PROGRAM IO_OP10A_10B_JB
VAR
	//INPUT
	WORD_AS_BIT_0: WORD_AS_BIT;
	WORD_AS_BIT_1: WORD_AS_BIT;
	WORD_AS_BIT_2: WORD_AS_BIT;
	WORD_AS_BIT_3: WORD_AS_BIT;	
	//OUTPUT
	BIT_AS_WORD_0: BIT_AS_WORD;
	BIT_AS_WORD_1: BIT_AS_WORD;
	BIT_AS_WORD_2: BIT_AS_WORD;
	BIT_AS_WORD_3: BIT_AS_WORD;	
	//OP10A JB DI/DO 
	OP10A_BOWL_FEEDER_JB_16DI_MODULE_1 AT %I* : WORD;
	OP10A_BOWL_FEEDER_JB_16DI_MODULE_2 AT %I* : WORD;
	OP10A_BOWL_FEEDER_JB_16DO_MODULE_1 AT %Q* : WORD;
	OP10A_BOWL_FEEDER_JB_16DO_MODULE_2 AT %Q* : WORD;
	//OP10B JB DI/DO 
	OP10B_BOWL_FEEDER_JB_16DI_MODULE_1 AT %I* : WORD;
	OP10B_BOWL_FEEDER_JB_16DI_MODULE_2 AT %I* : WORD;
	OP10B_BOWL_FEEDER_JB_16DO_MODULE_1 AT %Q* : WORD;
	OP10B_BOWL_FEEDER_JB_16DO_MODULE_2 AT %Q* : WORD;
END_VAR

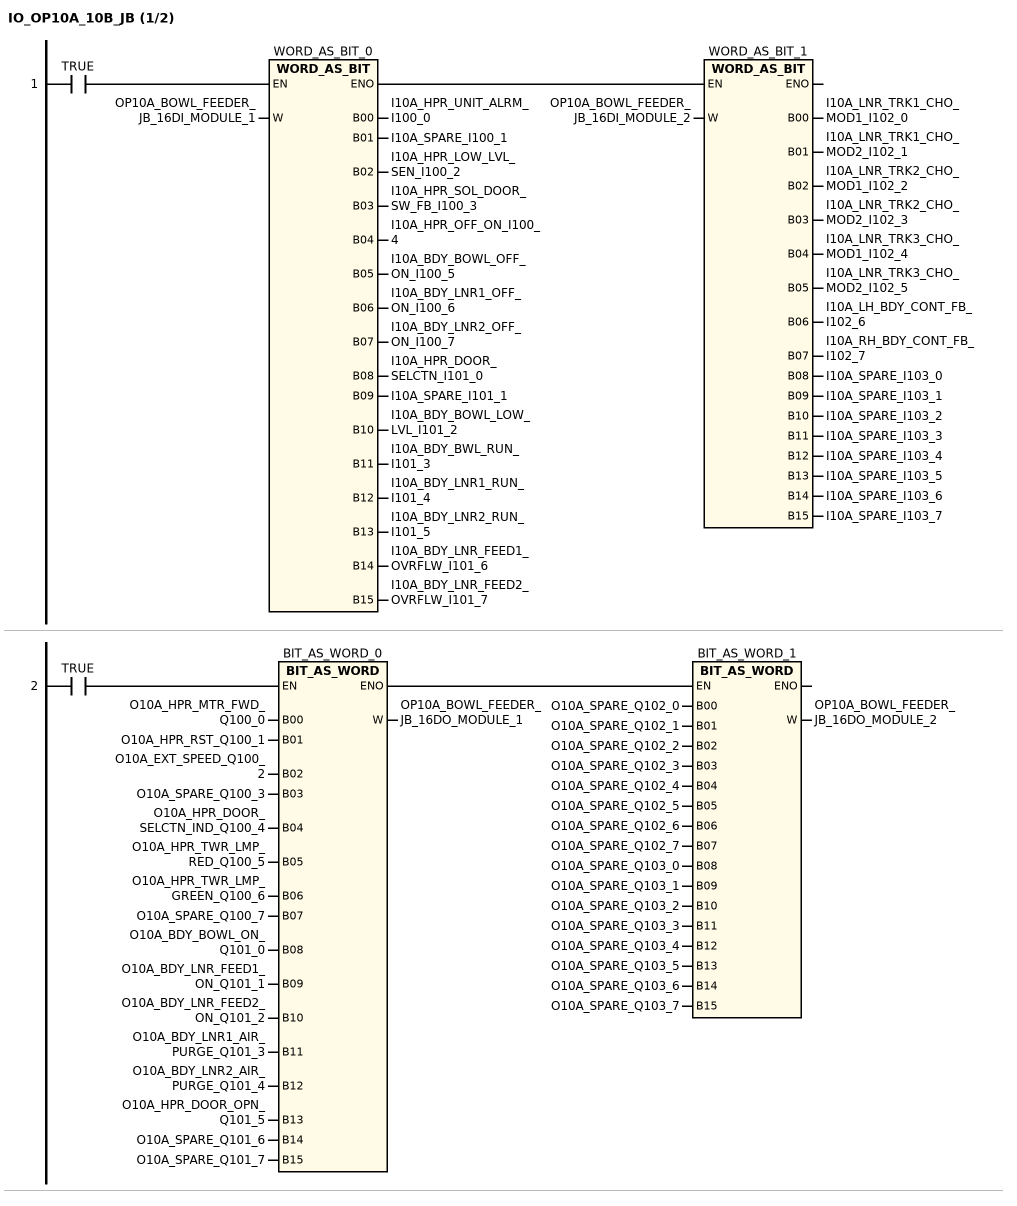
// NETWORK 1
WORD_AS_BIT_0(
    W := OP10A_BOWL_FEEDER_JB_16DI_MODULE_1,
    B00 => I10A_HPR_UNIT_ALRM_I100_0,
    B01 => I10A_SPARE_I100_1,
    B02 => I10A_HPR_LOW_LVL_SEN_I100_2,
    B03 => I10A_HPR_SOL_DOOR_SW_FB_I100_3,
    B04 => I10A_HPR_OFF_ON_I100_4,
    B05 => I10A_BDY_BOWL_OFF_ON_I100_5,
    B06 => I10A_BDY_LNR1_OFF_ON_I100_6,
    B07 => I10A_BDY_LNR2_OFF_ON_I100_7,
    B08 => I10A_HPR_DOOR_SELCTN_I101_0,
    B09 => I10A_SPARE_I101_1,
    B10 => I10A_BDY_BOWL_LOW_LVL_I101_2,
    B11 => I10A_BDY_BWL_RUN_I101_3,
    B12 => I10A_BDY_LNR1_RUN_I101_4,
    B13 => I10A_BDY_LNR2_RUN_I101_5,
    B14 => I10A_BDY_LNR_FEED1_OVRFLW_I101_6,
    B15 => I10A_BDY_LNR_FEED2_OVRFLW_I101_7); // WORD_AS_BIT
WORD_AS_BIT_1(
    W := OP10A_BOWL_FEEDER_JB_16DI_MODULE_2,
    B00 => I10A_LNR_TRK1_CHO_MOD1_I102_0,
    B01 => I10A_LNR_TRK1_CHO_MOD2_I102_1,
    B02 => I10A_LNR_TRK2_CHO_MOD1_I102_2,
    B03 => I10A_LNR_TRK2_CHO_MOD2_I102_3,
    B04 => I10A_LNR_TRK3_CHO_MOD1_I102_4,
    B05 => I10A_LNR_TRK3_CHO_MOD2_I102_5,
    B06 => I10A_LH_BDY_CONT_FB_I102_6,
    B07 => I10A_RH_BDY_CONT_FB_I102_7,
    B08 => I10A_SPARE_I103_0,
    B09 => I10A_SPARE_I103_1,
    B10 => I10A_SPARE_I103_2,
    B11 => I10A_SPARE_I103_3,
    B12 => I10A_SPARE_I103_4,
    B13 => I10A_SPARE_I103_5,
    B14 => I10A_SPARE_I103_6,
    B15 => I10A_SPARE_I103_7); // WORD_AS_BIT

// NETWORK 2
BIT_AS_WORD_0(
    B00 := O10A_HPR_MTR_FWD_Q100_0,
    B01 := O10A_HPR_RST_Q100_1,
    B02 := O10A_EXT_SPEED_Q100_2,
    B03 := O10A_SPARE_Q100_3,
    B04 := O10A_HPR_DOOR_SELCTN_IND_Q100_4,
    B05 := O10A_HPR_TWR_LMP_RED_Q100_5,
    B06 := O10A_HPR_TWR_LMP_GREEN_Q100_6,
    B07 := O10A_SPARE_Q100_7,
    B08 := O10A_BDY_BOWL_ON_Q101_0,
    B09 := O10A_BDY_LNR_FEED1_ON_Q101_1,
    B10 := O10A_BDY_LNR_FEED2_ON_Q101_2,
    B11 := O10A_BDY_LNR1_AIR_PURGE_Q101_3,
    B12 := O10A_BDY_LNR2_AIR_PURGE_Q101_4,
    B13 := O10A_HPR_DOOR_OPN_Q101_5,
    B14 := O10A_SPARE_Q101_6,
    B15 := O10A_SPARE_Q101_7,
    W => OP10A_BOWL_FEEDER_JB_16DO_MODULE_1); // BIT_AS_WORD
BIT_AS_WORD_1(
    B00 := O10A_SPARE_Q102_0,
    B01 := O10A_SPARE_Q102_1,
    B02 := O10A_SPARE_Q102_2,
    B03 := O10A_SPARE_Q102_3,
    B04 := O10A_SPARE_Q102_4,
    B05 := O10A_SPARE_Q102_5,
    B06 := O10A_SPARE_Q102_6,
    B07 := O10A_SPARE_Q102_7,
    B08 := O10A_SPARE_Q103_0,
    B09 := O10A_SPARE_Q103_1,
    B10 := O10A_SPARE_Q103_2,
    B11 := O10A_SPARE_Q103_3,
    B12 := O10A_SPARE_Q103_4,
    B13 := O10A_SPARE_Q103_5,
    B14 := O10A_SPARE_Q103_6,
    B15 := O10A_SPARE_Q103_7,
    W => OP10A_BOWL_FEEDER_JB_16DO_MODULE_2); // BIT_AS_WORD

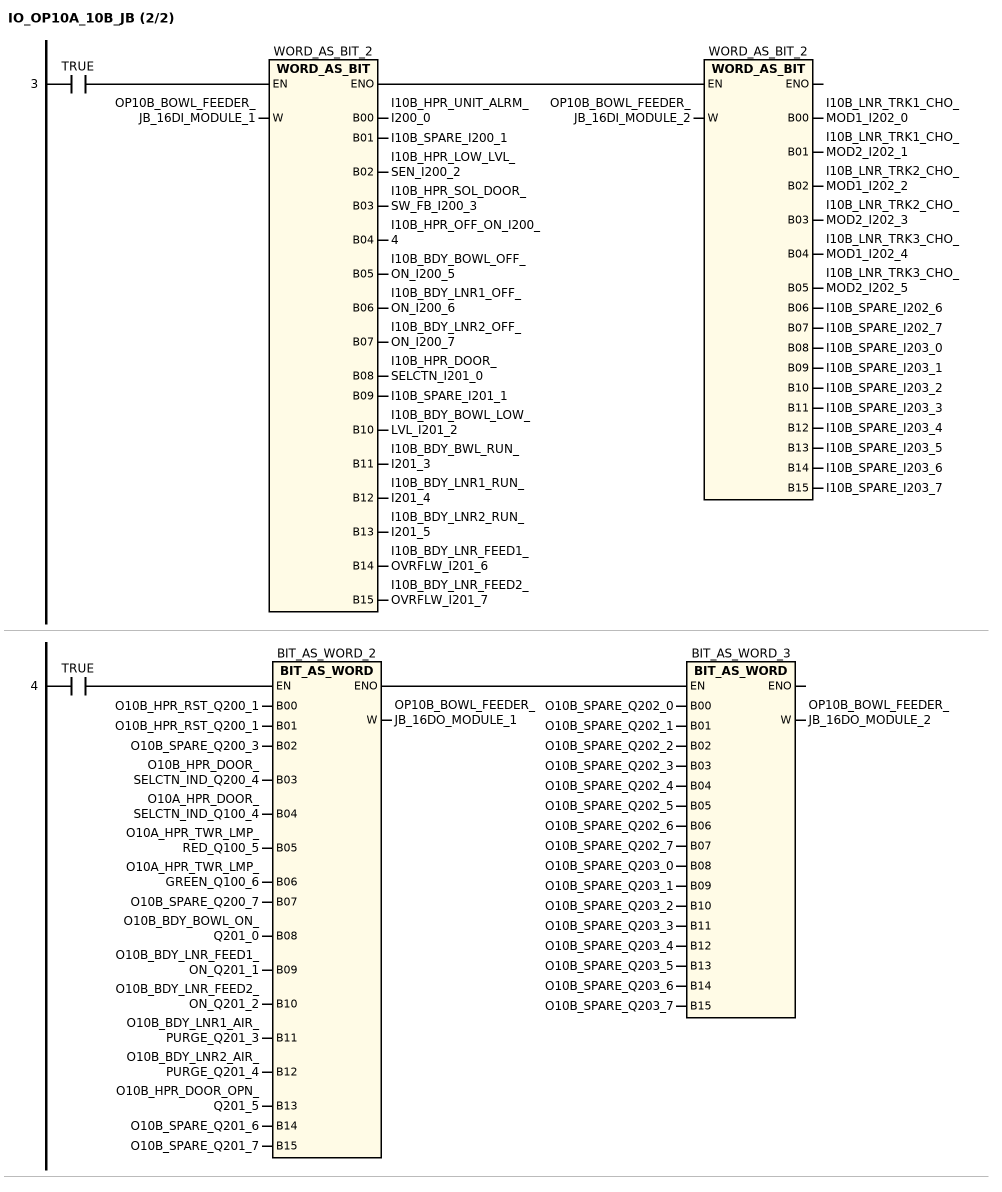
// NETWORK 3
WORD_AS_BIT_2(
    W := OP10B_BOWL_FEEDER_JB_16DI_MODULE_1,
    B00 => I10B_HPR_UNIT_ALRM_I200_0,
    B01 => I10B_SPARE_I200_1,
    B02 => I10B_HPR_LOW_LVL_SEN_I200_2,
    B03 => I10B_HPR_SOL_DOOR_SW_FB_I200_3,
    B04 => I10B_HPR_OFF_ON_I200_4,
    B05 => I10B_BDY_BOWL_OFF_ON_I200_5,
    B06 => I10B_BDY_LNR1_OFF_ON_I200_6,
    B07 => I10B_BDY_LNR2_OFF_ON_I200_7,
    B08 => I10B_HPR_DOOR_SELCTN_I201_0,
    B09 => I10B_SPARE_I201_1,
    B10 => I10B_BDY_BOWL_LOW_LVL_I201_2,
    B11 => I10B_BDY_BWL_RUN_I201_3,
    B12 => I10B_BDY_LNR1_RUN_I201_4,
    B13 => I10B_BDY_LNR2_RUN_I201_5,
    B14 => I10B_BDY_LNR_FEED1_OVRFLW_I201_6,
    B15 => I10B_BDY_LNR_FEED2_OVRFLW_I201_7); // WORD_AS_BIT
WORD_AS_BIT_2(
    W := OP10B_BOWL_FEEDER_JB_16DI_MODULE_2,
    B00 => I10B_LNR_TRK1_CHO_MOD1_I202_0,
    B01 => I10B_LNR_TRK1_CHO_MOD2_I202_1,
    B02 => I10B_LNR_TRK2_CHO_MOD1_I202_2,
    B03 => I10B_LNR_TRK2_CHO_MOD2_I202_3,
    B04 => I10B_LNR_TRK3_CHO_MOD1_I202_4,
    B05 => I10B_LNR_TRK3_CHO_MOD2_I202_5,
    B06 => I10B_SPARE_I202_6,
    B07 => I10B_SPARE_I202_7,
    B08 => I10B_SPARE_I203_0,
    B09 => I10B_SPARE_I203_1,
    B10 => I10B_SPARE_I203_2,
    B11 => I10B_SPARE_I203_3,
    B12 => I10B_SPARE_I203_4,
    B13 => I10B_SPARE_I203_5,
    B14 => I10B_SPARE_I203_6,
    B15 => I10B_SPARE_I203_7); // WORD_AS_BIT

// NETWORK 4
BIT_AS_WORD_2(
    B00 := O10B_HPR_RST_Q200_1,
    B01 := O10B_HPR_RST_Q200_1,
    B02 := O10B_SPARE_Q200_3,
    B03 := O10B_HPR_DOOR_SELCTN_IND_Q200_4,
    B04 := O10A_HPR_DOOR_SELCTN_IND_Q100_4,
    B05 := O10A_HPR_TWR_LMP_RED_Q100_5,
    B06 := O10A_HPR_TWR_LMP_GREEN_Q100_6,
    B07 := O10B_SPARE_Q200_7,
    B08 := O10B_BDY_BOWL_ON_Q201_0,
    B09 := O10B_BDY_LNR_FEED1_ON_Q201_1,
    B10 := O10B_BDY_LNR_FEED2_ON_Q201_2,
    B11 := O10B_BDY_LNR1_AIR_PURGE_Q201_3,
    B12 := O10B_BDY_LNR2_AIR_PURGE_Q201_4,
    B13 := O10B_HPR_DOOR_OPN_Q201_5,
    B14 := O10B_SPARE_Q201_6,
    B15 := O10B_SPARE_Q201_7,
    W => OP10B_BOWL_FEEDER_JB_16DO_MODULE_1); // BIT_AS_WORD
BIT_AS_WORD_3(
    B00 := O10B_SPARE_Q202_0,
    B01 := O10B_SPARE_Q202_1,
    B02 := O10B_SPARE_Q202_2,
    B03 := O10B_SPARE_Q202_3,
    B04 := O10B_SPARE_Q202_4,
    B05 := O10B_SPARE_Q202_5,
    B06 := O10B_SPARE_Q202_6,
    B07 := O10B_SPARE_Q202_7,
    B08 := O10B_SPARE_Q203_0,
    B09 := O10B_SPARE_Q203_1,
    B10 := O10B_SPARE_Q203_2,
    B11 := O10B_SPARE_Q203_3,
    B12 := O10B_SPARE_Q203_4,
    B13 := O10B_SPARE_Q203_5,
    B14 := O10B_SPARE_Q203_6,
    B15 := O10B_SPARE_Q203_7,
    W => OP10B_BOWL_FEEDER_JB_16DO_MODULE_2); // BIT_AS_WORD

END_PROGRAM

(* stored: Version 1.1.0.1, ProductVersion 3.1.4024.11
   POU IO_OP10A_10B_JB: Id {efaefa1e-d41a-431f-a118-e246a40978aa}, SpecialFunc None *)
